// TIA Portal V19 export
ORGANIZATION_BLOCK "CYC_INT1"   // OB35, STL, CyclicInterrupt
TITLE = "Cylic Interupt, 100ms
{ S7_Optimized_Access := 'TRUE' }
VERSION : 0.0
// stored: AutoNumber false
   VAR_INPUT
      Initial_Call : Bool;   // Initial call of this OB
      Event_Count : Int;   // Events discarded
   END_VAR
   VAR_TEMP
      t_dint : DInt;
      t_real : Real;
   END_VAR
BEGIN

NETWORK
TITLE = PID - Controller
// PID-Regulator for Steam Valve 01.57
      CALL  "STD_PID_CONTROL"
      ( AUTOMATIC := "AutoTT0172/IP0157",
        MANUAL    := "ManTT0172/IP0157",
        ADAPT     := FALSE,
        DIRECT    := FALSE,  //HEATER
        PV        := "MeasuredValues".TT0172REAL,  //"DB-ANALOG INPUT".TT0172REAL
        SP        := "PID_TT0172/IP0157".TT0172SpDBD,
        FF        := 0.0,
        PV_MAX    := 1600.0,
        PV_MIN    := 0.0,
        OP_MAX    := 10000.0,
        OP_MIN    := 0.0,
        P         := "PID_TT0172/IP0157".IP0157PPID,
        I         := "PID_TT0172/IP0157".IP0157IPID,
        D         := "PID_TT0172/IP0157".IP0157DPID,
        ScanTime  := 0.1,
        OP        := "PID_TT0172/IP0157".IP0157OuPID,
        intgr     := "PID_TT0172/IP0157".IP0157IntPID,
        diff      := "PID_TT0172/IP0157".IP0157DifPID,
        ndev_1    := "PID_TT0172/IP0157".IP0157DevPID
      );


      CALL  "MonitoringValves", "MonitoringValves_DB";


      A     "MM0139";  // 4 mA TO IP 01.57 IF PUMP FB MISSING
      AN    "M0139S";
      JC    FAUL;
      JC    END;
FAUL: L     0;
      T     "PID_TT0172/IP0157".IP0157OuPID;
END:  NOP   0;

// Set up M09.40 PID Loop PV's
      L     "PG_Devices".PTX0941.Value_p;
      T     "M0940_PIDInterfaceDB".PC.PV;

      L     "hf HoperLevelF2";
      T     #t_dint;
      DTR;
      T     "M0940_PIDInterfaceDB".LC.PV;

      L     "Max_F2";
      L     "Min_F2";
      -I;
      T     #t_dint;
      DTR;
      L     0.1;
      *R;
      T     #t_real;
      L     "Max_F2";
      T     #t_dint;
      DTR;
      L     #t_real;
      -R;
      T     "M0940_PIDInterfaceDB".LC.SP;


      CALL  "PID HMI Interface", "PID_Loops_DB"
      ( LoopSelection := ,
        RPM           := ,
        Hmi           := "PIDHmiInterfaceDB".M0940,
        PC            := "M0940_PIDInterfaceDB".PC,
        LC            := "M0940_PIDInterfaceDB".LC
      );











END_ORGANIZATION_BLOCK
